KUKA KRL program: wenglorUserConfig.src, wenglorUserConfig.dat

--- wenglorUserConfig.src ---
&ACCESS RVO
&REL 23
&PARAM EDITMASK = *
DEF wenglorUserConfig( )
   ;**************************************
   ;
   ; Module: wenglorUserConfig
   ; Author: wenglor sensoric GmbH
   ; Version: 2.1.0
   ;
   ; Description:
   ;   The file manages all user
   ;   configurations.
   ;
   ;**************************************
   ;FOLD INI;%{PE}
      ;FOLD BASISTECH INI
         GLOBAL INTERRUPT DECL 3 WHEN $STOPMESS==TRUE DO IR_STOPM ( )
         INTERRUPT ON 3
         BAS (#INITMOV,0 )
      ;ENDFOLD (BASISTECH INI)
      ;FOLD USER INI
         ;Make your modifications here

      ;ENDFOLD (USER INI)
   ;ENDFOLD (INI)
   ;----------------------------------------
   ;----------------------------------------
   ; Name of the xml file
   W_CONNECTION[] = "wenglorVision"
   ;----------------------------------------
   ;----------------------------------------
   ; Comment out the correct line depending
   ; on the selected camera/robot setup
   W_USE_CASE[] = "camera_not_on_robot"
   ;W_USE_CASE[] = "camera_on_robot"
   ;----------------------------------------
   ;----------------------------------------
   ; Comment out the correct line depending
   ; on the selected calibration board
   W_CALIBRATION_TARGET[] = "zvzj001"
   ;W_CALIBRATION_TARGET[] = "zvzj002"
   ;W_CALIBRATION_TARGET[] = "zvzj003"
   ;W_CALIBRATION_TARGET[] = "zvzj004"
   ;----------------------------------------
   ;----------------------------------------
   ; Define the uniVision jobs
   W_CALIBRATION_JOB[] = "calibration.u3p"
   W_DETECT_OBJECTS_JOB[] = "find_objects.u3p"
   W_DETECT_TARGET_JOB[] = "find_target.u3p"
   ;----------------------------------------
   ;----------------------------------------
   ; Adjust validation z safety offset [mm]
   W_SAFETY_OFFSET_MM = 10;
   ;----------------------------------------
   ;----------------------------------------
   ; Adjust the number of calibration poses
   ; you want to use. 5 poses are required
   ; at least.
   W_NUM_CALIBRATION_POSES = 5
   ;----------------------------------------
   ;----------------------------------------
   ; Comment out the correct line depending
   ; on the selected detection
   W_USER_COMMAND[] = "singleDetection"
   ;W_USER_COMMAND[] = "multiDetection"
   ;W_USER_COMMAND[] = "updateReferenceFrame"
   ;----------------------------------------
   ;----------------------------------------
   ; Mobile Platform use case:
   ; Adjust W_BASE_NUM and W_BASE_NAME in case of
   ; using updateReferenceFrame
   W_BASE_NUM = 10
   W_BASE_NAME[] = "wReferenceFrame"
   ; Set to TRUE after teaching the poses
   ; with the updated reference frame
   W_MACHINE_POSES_TAUGHT = FALSE
   ;----------------------------------------
   ;----------------------------------------
END

GLOBAL DEF moveTocalibrationPose(poseNum:IN)
   INT poseNum
   SWITCH poseNum
      CASE 1
         ; Add movement to calibration pose 1 here.
         ;

      CASE 2
         ; Add movement to calibration pose 2 here.
         ;

      CASE 3
         ; Add movement to calibration pose 3 here.
         ;

      CASE 4
         ; Add movement to calibration pose 4 here.
         ;

      CASE 5
         ; Add movement to calibration pose 5 here.
         ;

         ;------------------------------------
         ;------------------------------------
         ; Add more poses by copy "CASE #" and
         ; increase the pose number e.g.: CASE 6
         ; Make sure g_num_calibration_poses
         ; above has the right value.
         ;

      DEFAULT
         ; no movement
   ENDSWITCH

END

GLOBAL DEF moveToDetectObjectsPose()
   ; Add movement to detectObjectsPose here.
   ;

END

GLOBAL DEF moveToSafetyPose()
   ; Add movement to pose here.
   ; use case camera not on robot
   ; for removing calibration board
   ;

END

GLOBAL DEF moveToDetectTargetPose()
   ; Add movement to targetPose here.
   ;

END

GLOBAL DEF moveTo(pose:IN)
   DECL FRAME pose
   $VEL.CP = 0.1
   LIN pose
END

GLOBAL DEF testCalibrationPoses()
   INT i
   FOR i=1 to W_NUM_CALIBRATION_POSES
      moveTocalibrationPose(i)
   ENDFOR
END

--- wenglorUserConfig.dat ---
&ACCESS RV1
&REL 5
&PARAM EDITMASK = *
&PARAM TEMPLATE = C:\KRC\Roboter\Template\vorgabe
DEFDAT  wenglorUserConfig
   ;**************************************
   ;
   ; Module: wenglorUserConfig
   ; Author: wenglor sensoric GmbH
   ; Version: 2.0.0
   ;
   ; Description:
   ;   The file manages all user
   ;   configurations.
   ;
   ;**************************************
   ;FOLD EXTERNAL DECLARATIONS;%{PE}%MKUKATPBASIS,%CEXT,%VCOMMON,%P
   ;FOLD BASISTECH EXT;%{PE}%MKUKATPBASIS,%CEXT,%VEXT,%P
   EXT  BAS (BAS_COMMAND  :IN,REAL  :IN )
   DECL INT SUCCESS
   ;ENDFOLD (BASISTECH EXT)
   ;FOLD USER EXT;%{E}%MKUKATPUSER,%CEXT,%VEXT,%P
   ;Make your modifications here

   ;ENDFOLD (USER EXT)
   ;ENDFOLD (EXTERNAL DECLARATIONS)
ENDDAT
